# B&R Automation Studio project PLC_Eksamens_Projekt
Automation Studio 4.5.2.102

## Configuration Config1

CPU X20CP1382, AutomationRuntime D4.52, Build 4.1.2, Vc V4.52.0

### Hardware
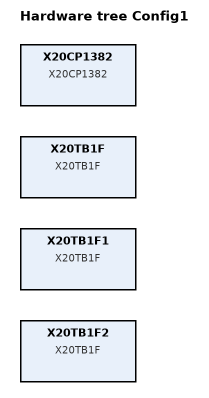
```
X20CP1382 : X20CP1382 v1.7.0.0  [X1 -> X1.SL; X2 -> X2.SL; X3 -> X3.SL]
  Module X1 (Type=X1, Virtual=true, Version=1.7.0.0)
    Connection (Connector=SS1, TargetModule=X20TB1F, TargetConnector=SS)
    Connection (Connector=SL, TargetModule=X20CP1382, TargetConnector=X1)
  Module X2 (Type=X2, Virtual=true, Version=1.7.0.0)
    Connection (Connector=SS1, TargetModule=X20TB1F1, TargetConnector=SS)
    Connection (Connector=SL, TargetModule=X20CP1382, TargetConnector=X2)
  Module X3 (Type=X3, Virtual=true, Version=1.7.0.0)
    Connection (Connector=SS1, TargetModule=X20TB1F2, TargetConnector=SS)
    Connection (Connector=SL, TargetModule=X20CP1382, TargetConnector=X3)
  Connector IF2:
    ActivateDevice = 1
  ConfigurationID = PLC_Eksamens_Projekt_Config1
  Simulation = 1
  SimulationInaPort = 11169
X20TB1F : X20TB1F v1.0.0.0
X20TB1F1 : X20TB1F v1.0.0.0
X20TB1F2 : X20TB1F v1.0.0.0
```

## Logical view

### Program Logical/Program

#### Types.typ
```iecst
(*Denne Type er de 3 stadier som vores robot arm kan befinde sig i.*)

TYPE
	RobotArm : 	STRUCT
		Placing : BOOL;
		Getting : BOOL;
	END_STRUCT;
END_TYPE
```

#### Variables.var
```iecst
VAR
	pos2OutOfPlace : BOOL;
	pos1OutOfPlace : BOOL;
	goBtn : BOOL;
	Eater : BOOL;
	convStart : BOOL;
	convStop : BOOL;
	robotToPos2 : BOOL;
	robotToPos1 : BOOL;
	pickerRobotRight : RobotArm;
	pickerRobotLeft : RobotArm;
	SorterRobot : RobotArm;
	PickerSpot : BOOL;
	ForPicking : f_trig;
END_VAR
```

#### Main.st
```iecst
PROGRAM _INIT
	(* Init værdier for alt i programmet *)

	goBtn := FALSE; // input fra experior
	pos1OutOfPlace := FALSE; // input fra experior weight 1
	pos2OutOfPlace := FALSE; // input fra experior weight 2
	convStart := FALSE; // output til experior
	convStop := FALSE; // output til experior
	robotToPos1 := FALSE; // output til robot
	robotToPos2 := FALSE; // output til robot

END_PROGRAM

PROGRAM _CYCLIC
	(* Go knappen som starter hele programmet*)
	IF goBtn = TRUE THEN
		convStart := TRUE;

	ELSE
		convStop := TRUE;
	END_IF;
	(*Hvis der trykkes stop eller bliver sendt stop signal skal båndet stoppe.*)
	IF convStop = TRUE THEN
		convStart := FALSE;
	END_IF;
	IF pos1OutOfPlace = TRUE AND pos2OutOfPlace = FALSE THEN
		robotToPos1 := TRUE;
		IF SorterRobot.Placing = TRUE AND Eater = TRUE THEN
			SorterRobot.Placing := FALSE;
		END_IF;
	END_IF;
	IF pos2OutOfPlace = TRUE AND pos1OutOfPlace = FALSE THEN

			robotToPos2 := TRUE;
			IF SorterRobot.Placing = TRUE AND Eater = TRUE THEN
			SorterRobot.Placing := FALSE;
		END_IF;
	END_IF;
	IF pos2OutOfPlace = TRUE AND pos1OutOfPlace = TRUE THEN
		convStop := TRUE;
		robotToPos1 := TRUE;
		IF SorterRobot.Placing = TRUE AND Eater = TRUE THEN
			robotToPos2 := TRUE;
			SorterRobot.Placing := FALSE;
		END_IF;

	END_IF;
			END_PROGRAM

			PROGRAM _EXIT
			(* Insert code here *)

			END_PROGRAM
```
